        1: // Current state (1=BUSY, 6=IDLE)
            GVL_Serial.stPumpStatus[nParsedAxis].CurrentState := STRING_TO_INT(sToken);
            GVL_Serial.stPumpStatus[nParsedAxis].IsBusy := (GVL_Serial.stPumpStatus[nParsedAxis].CurrentState = 1);
            GVL_Serial.stPumpStatus[nParsedAxis].IsIdle := (GVL_Serial.stPumpStatus[nParsedAxis].CurrentState = 6);

        2: // Volume remaining (ul) - raw value has offset, calculate corrected
            GVL_Serial.stPumpStatus[nParsedAxis].VolumeRemaining := STRING_TO_LREAL(sToken);
            // Correct offset using per-axis full reference point
            // Axis 0: Full=5000, Axis 1: Full=10000 (configurable in GVL_Serial.rFullReference)
            // Corrected = Raw + (SyringeSize - FullReference) so Full=SyringeSize, Empty=0
            GVL_Serial.stPumpStatus[nParsedAxis].VolumeRemainingCorrected :=
                GVL_Serial.stPumpStatus[nParsedAxis].VolumeRemaining +
                (GVL_Serial.rSyringeSize[nParsedAxis] - GVL_Serial.rFullReference[nParsedAxis]);

        3: // Syringe movements
            GVL_Serial.stPumpStatus[nParsedAxis].SyringeMovements := STRING_TO_DINT(sToken);

        4: // Cumulative volume (ul)
            GVL_Serial.stPumpStatus[nParsedAxis].CumulativeVolume := STRING_TO_LREAL(sToken);

        5: // Current flow rate (ul/min)
            GVL_Serial.stPumpStatus[nParsedAxis].CurrentFlowRate := STRING_TO_LREAL(sToken);

        6: // Node sensor 1
            GVL_Serial.stPumpStatus[nParsedAxis].NodeSensor1 := sToken;

        7: // Node sensor 2
            GVL_Serial.stPumpStatus[nParsedAxis].NodeSensor2 := sToken;

        8: // Total cumulative volume (firmware 1.4.26+)
            GVL_Serial.stPumpStatus[nParsedAxis].TotalCumulativeVol := STRING_TO_LREAL(sToken);
    END_CASE

    nFieldIndex := nFieldIndex + 1;

    // Safety limit - don't parse more than expected fields
    IF nFieldIndex > 9 THEN
        EXIT;
    END_IF
END_WHILE

// Mark as valid if we got at least the required fields (error, state, etc.)
GVL_Serial.stPumpStatus[nParsedAxis].Valid := (nFieldIndex >= 6);
END_ACTION

END_PROGRAM
